SEGMENT_TYPE Ethernet (* Ethernet Segment *)
  (* Standard: 61499 ITA; Description: Ethernet ... *)
  (* Version 0.1, 2008-06-02, GEBENH, Profactor GmbH *)
  (* Compiler header: abc.xyz *)
  (* Compiler classdef: Ethernet .... *)
  (* Compiler Java IBM VisualAge 3.0 *)
  VAR_INPUT
    Param : WSTRING; (* Param *)
  END_VAR
END_SEGMENT_TYPE
